TYPE ST_DoorsNLocks_get :
STRUCT
	b_ClientpanelDoorClosed			: BOOL;
	b_ControlPanelDoorClosed		: BOOL;	
END_STRUCT
END_TYPE

(* stored: Version 1.1.0.1, ProductVersion 3.1.4024.12
   DUT ST_DoorsNLocks_get: Id {5236b545-1465-4c3a-8495-06143d67e04c} *)
